Yaskawa INFORM job: R1_ROBOTCALIB.JBI

/JOB
//NAME R1_ROBOTCALIB
///FOLDERNAME INNE
//POS
///NPOS 8,8,0,0,0,0
///TOOL 0
///POSTYPE PULSE
///PULSE
C00000=-79435,66526,91949,-87641,27850,44418
C00001=-113840,23124,44283,-37571,7809,17460
C00002=-113840,7039,-16249,-8244,35523,3840
C00003=-80284,35755,10944,-42162,44072,20040
C00004=-27876,-43237,-7229,-75376,63305,45633
C00005=-91659,-102567,-30557,-120522,22322,58326
C00006=-91659,-159010,-96337,-90316,19631,43954
C00007=-28526,-67927,-67181,-66060,71620,34292
BC00000=397782,129,502200
BC00001=397782,129,502200
BC00002=397782,129,502200
BC00003=397782,129,502200
BC00004=397782,129,502200
BC00005=397782,129,502200
BC00006=397782,129,502200
BC00007=397782,129,502200
//INST
///DATE 2023/10/04 15:16
///ATTR SC,RW
///GROUP1 RB1,BS1
NOP
MOVJ C00000 BC00000 VJ=0.78 PL=0
MOVJ C00001 BC00001 VJ=0.78 PL=0
MOVJ C00002 BC00002 VJ=0.78 PL=0
MOVJ C00003 BC00003 VJ=0.78 PL=0
MOVJ C00004 BC00004 VJ=0.78 PL=0
MOVJ C00005 BC00005 VJ=0.78 PL=0
MOVJ C00006 BC00006 VJ=0.78 PL=0
MOVJ C00007 BC00007 VJ=0.78 PL=0
END
